FUNCTION_BLOCK FB_CRYO_EVAC_PDS EXTENDS FB_CRYO_EVAC_BASE
VAR_INPUT
END_VAR
VAR_OUTPUT
END_VAR
VAR
	rp:	FB_CRYO_PUMP_MVP030;	// Roughing Pump
	tp:	FB_CRYO_PUMP_HIPACE30;	// Turbo Molecular Pump
	
END_VAR

SUPER^();

METHOD M_Configure
VAR_INPUT
END_VAR
//
// Specific PDS IR Imager configuration.
//
IF NOT stat.bConfigured	THEN
	// MANDATORY: Set References !!!
	// If not done, system will crash !!!
	rpRef	REF=rp;
	tpRef	REF=tp;
	

	// Specific instance configuration, e.g. anything different
	// from the default values given in the cfg structure of type T_CRYO_EVAC_CFG.
	cfg.nPressGaugeType1	:= E_CRYO_SENSOR_TYPE_PRESS.PKR_360;
	cfg.nPressGaugeType2	:= E_CRYO_SENSOR_TYPE_PRESS.PKR_360;

	cfg.lrThld_Prevac := 5.0;	// Prevacuum pressure threshold
	// Cryo pressure threshold to start Turbo Pump before opening Valve
	cfg.lrThld_TP_SafeStartPressure := 0.01;	
	// Cryo pressure threshold to start Turbo Pump once Valve is open
	cfg.lrThld_Valve_SafeOpenPressure := 0.1;	
	
	cfg.tDelay := T#3S;	// Time delay before stopping Turbo Pump

	stat.bConfigured	:= TRUE;;
ELSE
	RETURN;	// Nothing to do any more
END_IF
END_METHOD

METHOD M_ExecuteControllers
VAR_INPUT
END_VAR
//
// Specific PDS IR Imager HW.
//

// Roughing Pump	
rp(	
	in_bSimulation	:= FALSE,
	in_sName		:= 'MVP 030',
	in_bEnable		:= ctrl.bEnable_RP,
	in_nModel		:= 30,
	in_bAutoMonitor	:= TRUE,
	in_nPeriod		:= 3000);

// Turbo Molecular Pump
tp(	
	in_bSimulation	:= FALSE,
	in_sName		:= 'HIPACE 30',
	in_bEnable		:= ctrl.bEnable_TP,
	in_nModel		:= 30,
	in_bAutoMonitor	:= TRUE,
	in_nPeriod		:= 3000);


valve(in_bEnable	:= ctrl.bEnable_Valve);
END_METHOD

END_FUNCTION_BLOCK

(* stored: Version 1.1.0.1, ProductVersion 3.1.4024.10
   POU FB_CRYO_EVAC_PDS: Id {770ab621-e26e-4156-9ff6-0b29338e8fc1}, SpecialFunc None
   Method M_Configure: Id {c81ffccd-8665-4123-a26c-ac1ffb1ce34a}
   Method M_ExecuteControllers: Id {f065ddb5-6f56-41ed-a017-ad71c793aae9} *)
